DATA_BLOCK "DB_RecipeMaster"
{ S7_Optimized_Access := 'TRUE' }
VERSION : 0.1
// ATTRIBUTES
// AUTO_NUMBER = False
// BLOCK_NUMBER = 2700
// END_ATTRIBUTES
   VAR
      Header : "UDT_RecipeHeader";
      SubProcess : Array[1..32] of "UDT_SubProcessRecipe";
      FixtureCodes : Array[1..16] of String[128];
      GripperCodes : Array[1..18] of String[128];
      VisionPrograms : Array[1..16] of Int;
   END_VAR


BEGIN
   Header.ProductName := 'Product_1';
   Header.ProductID := 'P1';
   Header.RecipeVersion := 'V1.0';
   Header.FixtureFamily := 1;
   Header.Enabled := TRUE;
   Header.CreatedBy := 'OP10';
   Header.UpdatedBy := 'OP10';
   Header.Comment := 'Seed recipe migrated from ST10_RecipeDB';

   FixtureCodes[1] := 'SZ23055-OP010-E-Compressor-ring1 Loading tooling-1';
   FixtureCodes[2] := 'SZ23055-OP010-E-Compressor-ring1 Loading tooling-2';
   FixtureCodes[3] := 'SZ23055-OP010-E-Compressor-ring1 Loading tooling-3';
   FixtureCodes[4] := 'SZ23055-OP010-E-Compressor-ring1 Loading tooling-4';
   FixtureCodes[5] := 'SZ23055-OP010-E-Compressor-ring1 Loading tooling-5';
   FixtureCodes[6] := 'SZ23055-OP010-E-Compressor-ring1 Loading tooling-6';
   FixtureCodes[7] := 'SZ23055-OP010-E-Compressor-ring1 Loading tooling-7';
   FixtureCodes[8] := 'SZ23055-OP010-E-Compressor-ring1 Loading tooling-8';
   FixtureCodes[9] := 'SZ23055-OP010-E-Compressor-ring2 Loading tooling-1';
   FixtureCodes[10] := 'SZ23055-OP010-E-Compressor-ring2 Loading tooling-2';
   FixtureCodes[11] := 'SZ23055-OP010-E-Compressor-ring2 Loading tooling-3';
   FixtureCodes[12] := 'SZ23055-OP010-E-Compressor-ring2 Loading tooling-4';

   GripperCodes[1] := 'SZ23055-OP010-E-Compressor-robot1 ring1 Left clamping jaw tooling-1';
   GripperCodes[2] := 'SZ23055-OP010-E-Compressor-robot1 ring1 Right clamping jaw tooling-2';
   GripperCodes[3] := 'SZ23055-OP010-E-Compressor-robot1 shaft Left clamping jaw tooling-1';
   GripperCodes[4] := 'SZ23055-OP010-E-Compressor-robot1 shaft Right clamping jaw tooling-2';
   GripperCodes[5] := 'SZ23055-OP010-E-Compressor-robot2 shaft Right clamping jaw tooling-2';
   GripperCodes[6] := 'SZ23055-OP010-E-Compressor-robot2 shaft Left clamping jaw tooling-1';

END_DATA_BLOCK

